PROGRAM Test
VAR
	State : INT := 0;
END_VAR

CASE State OF
	1:  Global.Tank1.Filling.ParamFillLevel := 1.8;
		Global.Tank1.Filling.Cmd.ManCtrl := TRUE;
		Global.Tank1.Filling.Cmd.StartMan:= TRUE;
		IF Global.Tank1.Filling.State.Done = TRUE THEN
			State := 2;
		END_IF
	2: //...
END_CASE

END_PROGRAM

(* stored: Version 1.1.0.1, ProductVersion 3.1.4024.12
   POU Test: Id {b48fe353-a43c-460a-bd31-5cbc20fa1301}, SpecialFunc None *)
